FUNCTION_BLOCK CAerationLogic_HMI (* Service Interface Function Block Type *)
  (* Standard: 61499-2 *)
  (* Version 0.0, 10/24/2023, SESA685388, Schneider Electric, template *)
  PACKAGE SE.Nereda;
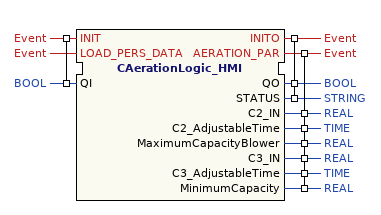
  EVENT_INPUT
    INIT WITH QI;
    LOAD_PERS_DATA;
  END_EVENT
  EVENT_OUTPUT
    INITO WITH QO, STATUS;
    AERATION_PAR WITH C2_IN, C3_IN, C2_AdjustableTime, C3_AdjustableTime, MaximumCapacityBlower, MinimumCapacity;
  END_EVENT
  VAR_INPUT
    QI : BOOL;
  END_VAR
  VAR_OUTPUT
    QO : BOOL; (* Event Output Qualifier *)
    STATUS : STRING; (* Service Status *)
    C2_IN : REAL;
    C2_AdjustableTime : TIME;
    MaximumCapacityBlower : REAL;
    C3_IN : REAL;
    C3_AdjustableTime : TIME;
    MinimumCapacity : REAL;
  END_VAR
  SERVICE /
    SEQUENCE 
    END_SEQUENCE
  END_SERVICE
END_FUNCTION_BLOCK
